PROGRAM SlaveArmControl
VAR
	// master robot data, input from master controller box
	m_masterRobotData AT %I* : MSCommu_MasterStatus;
	
	// all data from other tasks and controller 
	m_slaveInputDataPool : ST_SlaveInputDataPool;
		
	// slave robot data, ouput to master controller box
	m_slaveRobotData AT %Q* :MSCommu_slaveStatus;
	
	// slave robot status, including arm status and cartesian data, output to other tasks
	m_slaveStatus AT%Q* :ST_slaveStatus;
	
	// slave robot joint data, output to other tasks
	m_slaveJointsData AT %Q* :ST_slaveJointData;
	
	//slave motor in_output to safety check
	m_slaveMotorData AT %Q* : ST_slaveMotorData;
	
	//Electrical knife control code
	m_elecKnifeCtrlWordIO AT %Q* : DINT;
	
	// flag to init robot
	m_robotInit :BOOL :=FALSE;
	
	// wait time before robot init  for ethercat to be statble 
	m_robotInitWaitTime : LREAL:=0;
	m_armEtherCATOPTime : LREAL:=0;
	
	// slave robot
	m_slaveRobot:FB_SlaveRobot;

	// code execute time measure
	m_codeTime : Profiler;
	
	m_armIsDisable : ARRAY [1..4] OF BOOL;
	m_slaveCheckDetect : FB_MasterSlaveCheckDetect;
END_VAR

m_codeTime(START:=TRUE, RESET:=TRUE);
//check arms EtherCAT state is OP
IF NOT m_slaveInputDataPool.m_safetyData.m_armEtherCATAllOP AND NOT m_robotInit THEN
	m_armEtherCATOPTime := m_armEtherCATOPTime + g_slaveArmCtrlCycleTime;
	RETURN;
END_IF

// wait communication to be stable
IF(m_robotInitWaitTime<g_robotInitWaitTime) OR NOT(SafetyCheck.m_loadConfigFileOK) THEN
	m_robotInitWaitTime := m_robotInitWaitTime+g_slaveArmCtrlCycleTime;
	RETURN;
END_IF

// robot init
IF m_robotInit =FALSE THEN
	m_slaveRobot.Init();
	m_robotInit:=TRUE;
END_IF

// input from UI
UIInputProcess();

// master input data cast
masterInputDataCast(m_masterRobotData, m_slaveInputDataPool.m_masterStatus);

// robot run
m_slaveRobot.run(m_slaveInputDataPool);

// update data pool
m_slaveRobot.getStatus(m_slaveStatus,m_slaveMotorData,m_slaveJointsData);

// slave output data cast
slaveOutputDataCast(m_slaveInputDataPool.m_setupStatus, m_slaveStatus, m_slaveRobotData);

// output to UI
UIOutputProcess();

m_codeTime(START:=FALSE);

// convert from MSCommu_Mastertatus for master-slave communication to local ST_MasterStatus for control
METHOD masterInputDataCast : BOOL
VAR_IN_OUT CONSTANT
	masterInputData:MSCommu_MasterStatus;
END_VAR
VAR_IN_OUT
	masterStatus :ST_MasterStatus;
END_VAR

VAR
	i : INT;
END_VAR
masterStatus.m_masterHeartBeat := masterInputData.m_heartBeat;
masterStatus.m_motionScale := masterInputData.m_motionScale;
masterStatus.m_slaveSelfCheckFlag :=m_slaveCheckDetect.run(masterInputData.m_slaveSelfCheckFlag OR GVL_interactUI.g_salveSelfCheckEnable);
masterStatus.m_masterStopButton := masterInputData.m_masterStopButton;
masterStatus.m_uiResetFault := masterInputData.m_uiResetFault;
m_elecKnifeCtrlWordIO := masterInputData.m_elecKnifeCtrlWordIO;

FOR i:=1 TO g_mArmNum DO
	masterStatus.m_armState[i] := masterInputData.m_armState[i];
	masterStatus.m_teleSlaveArmIdx[i] :=masterInputData.m_teleSlaveArmIdx[i];
	masterStatus.m_gripAngle[i] := masterInputData.m_gripAngle[i];
	masterStatus.m_curArmPose[i].m_pos := masterInputData.m_curArmPose[i].m_pos;
	masterStatus.m_curArmPose[i].m_rot := masterInputData.m_curArmPose[i].m_rot;
	masterStatus.m_curArmTwist[i] :=masterInputData.m_curArmTwist[i];
	masterStatus.m_pedalHover[i] := masterInputData.m_pedalHover[i];
	masterStatus.m_electricKnifePedalTrigger[i] := masterInputData.m_electricKnifePedalTrigger[i];
	masterStatus.m_tryMSControl[i] := masterInputData.m_tryMSControl[i];
END_FOR
END_METHOD

// convert from local ST_SlaveStatus for control to MSCommu_SlaveStatus for master-slave communication
METHOD slaveOutputDataCast : BOOL
VAR_IN_OUT CONSTANT
	setupStatus :ST_SetupStatus;
	slaveStatus :ST_SlaveStatus;
END_VAR
VAR_IN_OUT 
	slaveOutputData : MSCommu_SlaveStatus;
END_VAR

VAR
	slavePoseInCart, slavePoseInScope:ST_Frame;
	tmpFrame :ST_Frame;
	forceBipolarMode : BOOL;
	scopeUpDown : UINT;
	i :INT;
END_VAR
// Slave heart beat
IF slaveOutputData.m_heartBeat > 10 THEN
	slaveOutputData.m_heartBeat :=0;
ELSE
	slaveOutputData.m_heartBeat :=slaveOutputData.m_heartBeat+1;
END_IF

FOR i := 1 TO g_sArmNum DO
	slaveOutputData.m_slaveAllowInMS :=((SlaveArmControl.m_slaveInputDataPool.m_UIData.m_slaveArmDisableFlag[i] OR SlaveArmControl.m_slaveRobot.m_panelMountedFlag[i]) AND  SafetyCheck.m_dumpEnergy > 30)
								OR m_slaveInputDataPool.m_UIData.m_masterSlaveFlag ;	
	IF NOT slaveOutputData.m_slaveAllowInMS THEN
		EXIT;
	END_IF
END_FOR


slaveOutputData.m_seflCheckPass:=  m_slaveInputDataPool.m_UIData.m_armSelfCheckFinshed[1] AND  m_slaveInputDataPool.m_UIData.m_armSelfCheckFinshed[2] AND m_slaveInputDataPool.m_UIData.m_armSelfCheckFinshed[3] AND m_slaveInputDataPool.m_UIData.m_armSelfCheckFinshed[4] ;
slaveOutputData.m_endoscopeMounted :=slaveStatus.m_endoscopeMounted;
slaveOutputData.m_endoscopePose.m_pos :=slaveStatus.m_endoscopePose.m_pos;
slaveOutputData.m_endoscopePose.m_rot :=slaveStatus.m_endoscopePose.m_rot;
slaveOutputData.m_slaveStopButton := NOT SafetyCheck.m_stopButton;
//clear value
slaveOutputData.m_publicByte := 0;
	
FOR i:= 1 TO g_sArmNum DO
	slaveOutputData.m_armState[i] := slaveStatus.m_armState[i];
	slaveOutputData.m_instruStauts[i].m_fingerAngle := slaveStatus.m_instruStauts[i].m_fingerAngle;
	slaveOutputData.m_instruStauts[i].m_ready := slaveStatus.m_instruStauts[i].m_ready;
	slaveOutputData.m_instruStauts[i].m_type := slaveStatus.m_instruStauts[i].m_type;
	slaveOutputData.m_instruEnergyType[i] := m_slaveRobot.m_slaveArms[i].m_instrument.instruTypeInfo.m_energyType;
	slavePoseInCart := transform(setupStatus.m_curEndPose[i], slaveStatus.m_curArmPose[i]);
	tmpFrame :=invFrame(slaveStatus.m_endoscopePose);
	slavePoseInScope := transform(tmpFrame, slavePoseInCart);
	slaveOutputData.m_curArmPose[i].m_pos :=slavePoseInScope.m_pos;
	slaveOutputData.m_curArmPose[i].m_rot :=slavePoseInScope.m_rot;
	slaveOutputData.m_masterSlavePoseError[i] :=slaveStatus.m_masterSlavePoseError[i];
	slaveOutputData.m_trocarOnFlag[i] := m_slaveRobot.m_slaveArms[i].trocarOn OR m_slaveRobot.m_instrumentMountedFlag[i];

	//public byte write
	forceBipolarMode := m_slaveRobot.m_slaveArms[i].instrument.forceBipolarMode AND m_slaveRobot.m_slaveArms[i].m_joints[4].m_motorInputs.m_statusWord = DriverStatusWord_OP;
	slaveOutputData.m_publicByte :=slaveOutputData.m_publicByte OR (SHL(TO_LINT(forceBipolarMode),i-1));
END_FOR
scopeUpDown := GVL_interactUI.g_uiReadScopeUpDown;
slaveOutputData.m_publicByte :=slaveOutputData.m_publicByte OR (SHL(TO_LINT(scopeUpDown),5));
END_METHOD

// tranform data from UI(global variable write by ADS) to ST_UIData
METHOD UIInputProcess : BOOL
VAR_INPUT
END_VAR
VAR
	i:int;
END_VAR
// arm disable
FOR i:=1 TO g_sArmNum DO 
	m_slaveInputDataPool.m_UIData.m_slaveArmDisableFlag[i]:= FALSE;
	
	IF GVL_interactUI.g_armIsDisable = i OR m_armIsDisable[i] THEN
		m_slaveInputDataPool.m_UIData.m_slaveArmDisableFlag[i]:= TRUE;
	END_IF
END_FOR


FOR i:=1 TO g_sArmNum DO 
	IF m_slaveRobot.m_slaveArmState[i] = SlaveArmState_MasterSlave THEN
		m_slaveInputDataPool.m_UIData.m_masterSlaveFlag :=TRUE;
	END_IF
END_FOR
END_METHOD

METHOD UIOutputProcess : BOOL
VAR_INPUT
END_VAR

VAR
	i , j: INT;
	teleSlaveArmIdx :ARRAY[1..g_mArmNum] OF E_MatchedSlaveArmIdx;
	masterslaveMode :BOOL;
END_VAR

VAR_STAT
	m_instruUsageCountsLast : ARRAY [1..g_sArmNum] OF ULINT;
END_VAR

//arm state machine
GVL_interactUI.g_armStateMachine.m_stateMachineArm1:=m_slaveStatus.m_armState[1];
GVL_interactUI.g_armStateMachine.m_stateMachineArm2:=m_slaveStatus.m_armState[2];
GVL_interactUI.g_armStateMachine.m_stateMachineArm3:=m_slaveStatus.m_armState[3];
GVL_interactUI.g_armStateMachine.m_stateMachineArm4:=m_slaveStatus.m_armState[4];

//arm is adjustment state
FOR i := 1 TO g_sArmNum BY 1 DO
	IF m_slaveStatus.m_armState[i] = SlaveArmState_Adjust OR m_slaveInputDataPool.m_setupStatus.m_armState[i] = SetupArmState_ManualAdjust 
							OR m_slaveInputDataPool.m_setupStatus.m_armState[i] = SetupArmState_AutoAdjust THEN
		GVL_interactUI.g_armIsAdjustment[i] := 1;
	ELSE
		GVL_interactUI.g_armIsAdjustment[i] := 0;
	END_IF
END_FOR


//arm self check status
FOR i := 1 TO g_sArmNum DO
	m_slaveInputDataPool.m_UIData.m_armInSelfCheck[i] := m_slaveStatus.m_armState[i] = SlaveArmState_SelfCheck AND NOT m_slaveInputDataPool.m_UIData.m_slaveArmDisableFlag[i];
	m_slaveInputDataPool.m_UIData.m_armSelfCheckFinshed[i] := m_slaveStatus.m_selfCheckPass[i] OR m_slaveInputDataPool.m_UIData.m_slaveArmDisableFlag[i];
END_FOR

IF m_slaveInputDataPool.m_UIData.m_armInSelfCheck[1] OR m_slaveInputDataPool.m_UIData.m_armInSelfCheck[2] OR m_slaveInputDataPool.m_UIData.m_armInSelfCheck[3] OR m_slaveInputDataPool.m_UIData.m_armInSelfCheck[4] THEN
	GVL_interactUI.g_slaveSelfCheckStatus := 1;
ELSIF m_slaveInputDataPool.m_UIData.m_armSelfCheckFinshed[1] AND m_slaveInputDataPool.m_UIData.m_armSelfCheckFinshed[2] AND m_slaveInputDataPool.m_UIData.m_armSelfCheckFinshed[3] AND m_slaveInputDataPool.m_UIData.m_armSelfCheckFinshed[4] THEN
	GVL_interactUI.g_slaveSelfCheckStatus := 2;
ELSE
	GVL_interactUI.g_slaveSelfCheckStatus := 0;
END_IF

//endoScope turn over enable
GVL_interactUI.g_scopeTurnOverEnable := FALSE;
FOR i := 1 TO g_sArmNum BY 1 DO
	IF m_slaveStatus.m_instruStauts[i].m_type = InstruType_Endoscope THEN
		GVL_interactUI.g_scopeTurnOverEnable := (m_slaveStatus.m_armState[i] = SlaveArmState_ScopeReady OR m_slaveStatus.m_armState[i] = SlaveArmState_PanelReady)
			AND NOT (m_slaveInputDataPool.m_setupStatus.m_armState[i]=SetupArmState_ManualAdjust);
		EXIT;
	END_IF
END_FOR
	

//instrument information export to UI
FOR i := 1 TO g_sArmNum DO
	GVL_interactUI.g_instruInformatiom[i].m_instruIsConnected:=m_slaveStatus.m_instruStauts[i].m_ready;
	GVL_interactUI.g_instruInformatiom[i].m_instruInMasterSlave := (m_slaveStatus.m_armState[i] = SlaveArmState_MasterSlave OR m_slaveStatus.m_armState[i] = SlaveArmState_EndoScope);
	IF m_slaveStatus.m_instruStauts[i].m_type = InstruType_Endoscope AND m_slaveRobot.m_instrumentMountedFlag[i] =TRUE THEN
		GVL_interactUI.g_instruInformatiom[i].m_instruType := 4;
		GVL_interactUI.g_scopeGravityAngle := m_slaveRobot.m_slaveArms[i].curDHJntPos[4];
	ELSE
		GVL_interactUI.g_instruInformatiom[i].m_instruType := m_slaveRobot.m_slaveArms[i].m_instrument.instruTypeInfo.m_energyType;
	END_IF
	
	GVL_interactUI.g_instruInformatiom[i].m_armId := i;
	GVL_interactUI.g_instruInformatiom[i].m_instruSerialNum :=  m_slaveRobot.m_slaveArms[i].m_instrument.onChipData.m_InstruseriesNum;
	GVL_interactUI.g_instruInformatiom[i].m_instruID := m_slaveRobot.m_slaveArms[i].m_instrument.instruType;
	GVL_interactUI.g_instruInformatiom[i].m_nameEn := m_slaveRobot.m_slaveArms[i].m_instrument.instruTypeInfo.m_instruName;
	GVL_interactUI.g_instruInformatiom[i].m_nameCh := m_slaveRobot.m_slaveArms[i].m_instrument.instruTypeInfo.m_instruNameCH;
	
	//instrument pedal hover and pedal active
	GVL_interactUI.g_instruInformatiom[i].m_pedalHover:=FALSE;
	GVL_interactUI.g_instruInformatiom[i].m_pedalActive := 0;
	GVL_interactUI.g_instruInformatiom[i].m_strongStatus:=m_slaveRobot.m_slaveArms[i].instrument.forceBipolarMode AND m_slaveRobot.m_slaveArms[i].m_joints[4].m_motorInputs.m_statusWord = DriverStatusWord_OP and m_slaveRobot.m_slaveArms[i].m_joints[4].m_motorOutputs.m_controlWord = DriverCtrlWord_OP;
	FOR j := 1 TO g_mArmNum BY 1 DO
		teleSlaveArmIdx[j] := m_slaveInputDataPool.m_masterStatus.m_teleSlaveArmIdx[j];
		 IF  teleSlaveArmIdx[j] > 0 AND teleSlaveArmIdx[j] <= 4  THEN
			IF m_slaveInputDataPool.m_masterStatus.m_pedalHover[j] = TRUE THEN
				GVL_interactUI.g_instruInformatiom[teleSlaveArmIdx[j]].m_pedalHover:=TRUE;
			ELSE
				GVL_interactUI.g_instruInformatiom[teleSlaveArmIdx[j]].m_pedalHover:=FALSE;
			END_IF
			GVL_interactUI.g_instruInformatiom[teleSlaveArmIdx[j]].m_pedalActive := m_slaveRobot.m_slaveArms[teleSlaveArmIdx[j]].updatePedalActive(teleSlaveArmIdx[j] , m_slaveInputDataPool.m_masterStatus.m_electricKnifePedalTrigger[j]);
		END_IF
	END_FOR
	
	//instrument number of  use
	IF m_slaveRobot.m_slaveArms[i].m_instrument.onChipData.m_InstruUsageCounts <> m_InstruUsageCountsLast[i] THEN
		GVL_interactUI.g_instruInformatiom[i].m_useLifeplc := ULINT_TO_UINT(m_slaveRobot.m_slaveArms[i].m_instrument.onChipData.m_InstruUsageCounts);
	END_IF
	m_InstruUsageCountsLast[i] :=m_slaveRobot.m_slaveArms[i].m_instrument.onChipData.m_InstruUsageCounts;
	
	//read-write instrument number of use
	m_slaveRobot.m_slaveArms[i].m_instrument.writeNumOfUseToChip(GVL_interactUI.g_instruInformatiom[i].m_useLifeplc + 1 =  GVL_interactUI.g_instruInformatiom[i].m_useLifeUi AND m_slaveRobot.m_slaveArms[i].m_instrument.onChipData.m_InstruReadSucceed, GVL_interactUI.g_instruInformatiom[i].m_useLifeUi);

	//intrument total number of use
	GVL_interactUI.g_instruInformatiom[i].m_instruTotalLife :=UDINT_TO_UINT( m_slaveRobot.m_slaveArms[i].m_instrument.m_maxUsageNum);
END_FOR

// instrument out-of-view information
masterslaveMode := FALSE;
FOR i := 1 TO g_sArmNum DO
	IF m_slaveStatus.m_armState[i] = SlaveArmState_masterSlave THEN
		masterslaveMode := TRUE;
		EXIT;
	END_IF
END_FOR
FOR i := 1 TO g_sArmNum DO
	IF masterslaveMode THEN
//	IF TRUE THEN
		GVL_interactUI.g_instruInformatiom[i].m_instruPosX:=0;
		GVL_interactUI.g_instruInformatiom[i].m_instruPosY:=0;
		GVL_interactUI.g_instruInformatiom[i].m_instruPosZ:=0;
	ELSE
		GVL_interactUI.g_instruInformatiom[i].m_instruPosX:=m_slaveInputDataPool.m_slaveDynaData.m_insruViewData[i][1];
		GVL_interactUI.g_instruInformatiom[i].m_instruPosY:=m_slaveInputDataPool.m_slaveDynaData.m_insruViewData[i][2];
		GVL_interactUI.g_instruInformatiom[i].m_instruPosZ:=m_slaveInputDataPool.m_slaveDynaData.m_insruViewData[i][3];
	END_IF
END_FOR

FOR i := 1 TO g_sArmNum DO
	GVL_IO.g_joint8IO[i][1] := m_slaveRobot.m_slaveArms[i].m_adjustOnFlag;
	GVL_IO.g_joint8IO[i][2] := SetupArmControl.m_setupRobot.m_setupArms[i].m_jnt5AdjustDir = 1;
	GVL_IO.g_joint8IO[i][3] := SetupArmControl.m_setupRobot.m_setupArms[i].m_jnt5AdjustDir = -1;
	GVL_IO.g_joint8IO[i][4] := SetupArmControl.m_setupRobot.m_setupArms[i].m_manualAdjustOnFlag;
	GVL_IO.g_joint8IO[i][5] := m_slaveRobot.m_slaveArms[i].m_trocarOnFlag;
	GVL_IO.g_jointPowerBoxIO[i][1] := (m_slaveRobot.m_slaveArms[i].m_panelInstrumentOnIO AND 10#4) = 4;
	GVL_IO.g_jointPowerBoxIO[i][2] := (m_slaveRobot.m_slaveArms[i].m_panelInstrumentOnIO AND 10#8) = 8;
	GVL_IO.g_jointPowerBoxIO[i][3] := (m_slaveRobot.m_slaveArms[i].m_panelInstrumentOnIO AND 10#1) = 1;
	GVL_IO.g_jointPowerBoxIO[i][4] := (m_slaveRobot.m_slaveArms[i].m_panelInstrumentOnIO AND 10#2) = 2;
	GVL_IO.g_jointPowerBoxIO[i][5] := (m_slaveRobot.m_slaveArms[i].m_panelInstrumentOnIO AND 10#64) = 64;
	GVL_IO.g_endoscopeSingle[i][1] := (m_slaveRobot.m_slaveArms[i].m_panelInstrumentOnIO AND 10#16) = 16;
	GVL_IO.g_endoscopeSingle[i][2] := (m_slaveRobot.m_slaveArms[i].m_panelInstrumentOnIO AND 10#32) = 32;
END_FOR
END_METHOD

END_PROGRAM

(* stored: Version 1.1.0.1, ProductVersion 3.1.4024.11
   POU SlaveArmControl: Id {6192c11b-cd6e-4883-b627-958acfb9caf3}, SpecialFunc None
   Method masterInputDataCast: Id {688f8323-8b5a-4cc7-b4b2-cb5f74424c3f}
   Method slaveOutputDataCast: Id {110717ec-abfc-4dc8-a3ed-d3c3fbcf321b}
   Method UIInputProcess: Id {9dd02246-5151-482e-a090-b6247e0a96d4}
   Method UIOutputProcess: Id {d0fa8c54-c1d5-4f7b-80a8-06c5ca1c6dd6} *)
